Staubli VAL3: onF1Event.pgx

program onF1Event()
  local bool l_bYes
  local string l_sMessage
  local string l_sPath
  local num l_nPath
  local string l_sButton[2]
  local string l_sPage
  local string l_sMode
begin
  // look if the bButton is enable
  if bButton[0]
    //
    //
    // do not active the simulation if cycle is active
    //
    if !cycleStatus:bCycle
      //
      call language:message(l_sMessage,214)
      // get the yes_no button Key
      call language:getYesNo(l_sButton)
      // ask the question
      call use:yes_no(l_sMessage,l_sButton,l_bYes)
      if l_bYes
        logMsg("[KERNEL] INTERFACE:Simulation of the program: "+sEvent)
        cycleStatus:iToSuperV.sType=sProgType
        cycleStatus:iToSuperV.sData=sEvent
        cycleStatus:nInterfaceToSV=2
        wait(cycleStatus:nInterfaceToSV==-1)
        // load the production page
        l_sMode="simulation"
        call loadPage("kernel/page/production",l_sMode)
        call use:setView(false)
        // logMsg
        logMsg("[KERNEL] INTERFACE:PAGE Select program")
      endIf
    endIf
  endIf
end
